Staubli VAL3: onRightEvent.pgx

program onRightEvent()
  local num l_nDefault
  local num i
begin
  //
  // right click
  //
  // select the next one
  //
  nProgID=(nProgID+1)%size(saveData:sProgType)
  if nProgID!=2
    sProgType=saveData:sProgType[nProgID]
  else
    sProgType=saveData:sProgType[0]
  endIf
  // load the progType
  call load()
  // rebuild the list
  call buildList()
  // refresh
  use:bUseRefresh=true
end
